SUBAPPLICATION Uebung_071b_AX (* WBSD auf UT ausgeben, Wegabhängige Impulse (Adapter Version) *)
  (* Standard: 61499-2; Description: Copyright (c) 2023-2026 Meisterschulen am Ostbahnhof This program and the accompanying materials are made available under the terms of the Eclipse Public License 2.0 which is available at https://www.eclipse.org/legal/epl-2.0/ SPDX-License-Identifier: EPL-2.0 *)
  (* Version 1.0, 2026-04-19, Franz Höpfinger, Meisterschulen am Ostbahnhof, initial API and implementation (Adapter Version of Uebung_071b) *)
  PACKAGE Uebungen;
  IMPORT Uebungen::const::UT::TECU::DefaultPool_TECU::NumberVariable_Wheel_based_machine_distance;
  IMPORT Uebungen::const::UT::TECU::DefaultPool_TECU::NumberVariable_Wheel_based_machine_speed;
  IMPORT logiBUS::io::DQ::logiBUS_DO::Output_Q1;
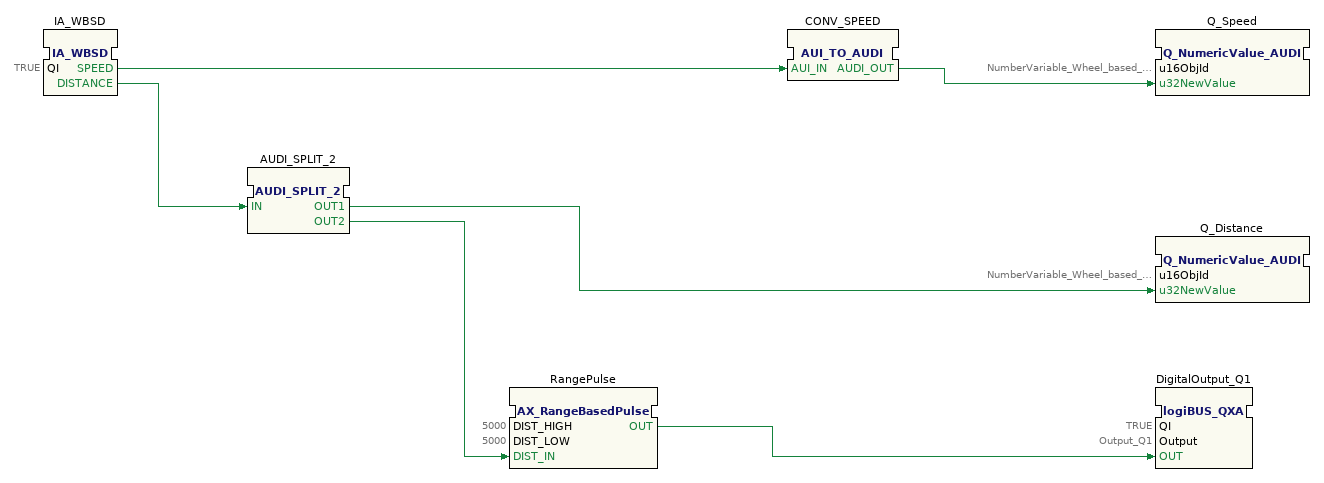
  (* Periodischer Puls alle 10 Meter (5m HIGH, 5m LOW) basierend auf Wegstrecke! *)
  FBS
    IA_WBSD : isobus::tecu::IA_WBSD(QI := TRUE);
    Q_Speed : isobus::UT::Q::Q_NumericValue_AUDI(u16ObjId := NumberVariable_Wheel_based_machine_speed);
    Q_Distance : isobus::UT::Q::Q_NumericValue_AUDI(u16ObjId := NumberVariable_Wheel_based_machine_distance);
    DigitalOutput_Q1 : logiBUS::io::DQ::logiBUS_QXA(QI := TRUE, Output := Output_Q1);
    RangePulse : logiBUS::signalprocessing::distance::AX_RangeBasedPulse(DIST_HIGH := 5000, DIST_LOW := 5000);
    CONV_SPEED : adapter::conversion::unidirectional::AUI_TO_AUDI;
    AUDI_SPLIT_2 : adapter::events::unidirectional::AUDI_SPLIT_2;
  END_FBS
  ADAPTER_CONNECTIONS
    IA_WBSD.SPEED TO CONV_SPEED.AUI_IN;
    CONV_SPEED.AUDI_OUT TO Q_Speed.u32NewValue;
    AUDI_SPLIT_2.OUT1 TO Q_Distance.u32NewValue;
    AUDI_SPLIT_2.OUT2 TO RangePulse.DIST_IN;
    RangePulse.OUT TO DigitalOutput_Q1.OUT;
    IA_WBSD.DISTANCE TO AUDI_SPLIT_2.IN;
  END_CONNECTIONS
END_SUBAPPLICATION
